/// Axis move additive parameter strucure
TYPE ST_AxisMoveAddParameter EXTENDS ST_AxisMoveParameter :
STRUCT
	/// Distance
	fDistance: LREAL;
END_STRUCT
END_TYPE

(* stored: Version 1.1.0.1, ProductVersion 3.1.4022.9
   DUT ST_AxisMoveAddParameter: Id {68fc6db6-27bb-48d3-b597-1859f1a8de77} *)
